(* Logix 5000 project; controller Hose_HP_Test_Rig_V1 vendor 1 type 14 code 149 rev 32.11; software revision 32.00; part 6 of 10 *)
(* tags used below, declared in another part *)
   BOTTOM_NOT_CLAMPED_STN3 : BOOL;
   FAIL_COMP_DROP_DEL : TIMER;
   FAIL_COMP_DROPPED : BOOL;
   FAIL_FLUSHED : DINT;
   FAULT_COMP_DROP_DEL : TIMER;
   FAULT_COMP_DROPPED : BOOL;
   FAULT_COMP_SENSOR : ALIAS FOR Local:2:I.Data.30;
   FAULT_FIFO_DEL : TIMER;
   FAULT_FLUSHED : DINT;
   FIFO_INDEX : DINT;
   FLUSH_BIN_DROP : TIMER;
   FLUSH_FAIL_BIN_DROP : TIMER;
   GET_FIRST_FAULTED : DINT;
   GOTO_FAIL_BIN_STN1 : DINT;
   GOTO_FAULT_BIN_STN3 : DINT;
   GOTO_FAULT_BIN_STN4 : DINT;
   ONS_100 : BOOL;
   ONS_101 : BOOL;
   ONS_102 : BOOL;
   ONS_70 : BOOL;
   ONS_76 : BOOL;
   ONS_77 : BOOL;
   ONS_78 : BOOL;
   ONS_79 : BOOL;
   ONS_80 : BOOL;
   ONS_81 : BOOL;
   ONS_82 : BOOL;
   ONS_83 : BOOL;
   ONS_84 : BOOL;
   ONS_85 : BOOL;
   ONS_86 : BOOL;
   ONS_87 : BOOL;
   ONS_88 : BOOL;
   ONS_89 : BOOL;
   ONS_90 : BOOL;
   ONS_91 : BOOL;
   ONS_92 : BOOL;
   ONS_93 : BOOL;
   ONS_95 : BOOL;
   ONS_96 : BOOL;
   ONS_97 : BOOL;
   ONS_98 : BOOL;
   ONS_99 : BOOL;
   TOP_NOT_CLAMPED_STN2 : BOOL;
   TOP_NOT_CLAMPED_STN3 : BOOL;
   TOP_NOT_CLAMPED_STN4 : BOOL;
   AUTO_TEST_ON_STN2 : BOOL;
   AUTO_TEST_ON_STN3 : BOOL;
   AUTO_TEST_ON_STN4 : BOOL;
   AUTO_TEST_SEL_STN1 : BOOL;
   AUTO_TEST_SEL_STN2 : BOOL;
   AUTO_TEST_SEL_STN3 : BOOL;
   AUTO_TEST_SEL_STN4 : BOOL;
   BOTTOM_CLAMP_2BPR_HIGH : BOOL;
   BOTTOM_CLAMP_2BPR_LOW : BOOL;
   BOTTOM_CLAMP_4BPR_HIGH : BOOL;
   BOTTOM_CLAMP_4BPR_LOW : BOOL;
   BOTTOM_CLAMP_4BPR_LOW_STN2 : BOOL;
   BOTTOM_CLAMP_PS_STN1 : ALIAS FOR Local:1:I.Data.13;
   BOTTOM_CLAMP_PS_STN2 : ALIAS FOR Local:2:I.Data.2;
   BOTTOM_CLAMP_PS_STN3 : ALIAS FOR Local:2:I.Data.7;
   BOTTOM_CLAMP_PS_STN4 : ALIAS FOR Local:2:I.Data.12;
   BOTTOM_NOT_CLAMPED_STN2 : BOOL;
   BOTTOM_NOT_CLAMPED_STN4 : BOOL;
   CHECK_TRACE_STS_STN2 : BOOL;
   CHECK_TRACE_STS_STN3 : BOOL;
   CHECK_TRACE_STS_STN4 : BOOL;
   COMP_FAULT_STN1 : BOOL;
   COMP_FAULT_STN2 : BOOL;
   COMP_FAULT_STN3 : BOOL;
   COMP_FAULT_STN4 : BOOL;
   CONS_FAIL_COUNT_STN1 : DINT;
   CONS_FAIL_COUNT_STN2 : DINT;
   CONS_FAIL_COUNT_STN3 : DINT;
   CONS_FAIL_COUNT_STN4 : DINT;
   CONS_FAIL_COUNTER_STN1 : COUNTER;
   CONS_FAIL_COUNTER_STN2 : COUNTER;
   CONS_FAIL_COUNTER_STN3 : COUNTER;
   CONS_FAIL_COUNTER_STN4 : COUNTER;
   CONS_FILL_HIGH_STN2 : BOOL;
   CONS_FILL_HIGH_STN3 : BOOL;
   CONS_FILL_HIGH_STN4 : BOOL;
   CONS_FILL_LOW_STN2 : BOOL;
   CONS_FILL_LOW_STN3 : BOOL;
   CONS_FILL_LOW_STN4 : BOOL;
   CONS_TEST_ON : BOOL;
   CONSTRICTION_CALB_SEL_STN1 : BOOL;
   CONSTRICTION_CALB_SEL_STN2 : BOOL;
   CONSTRICTION_CALB_SEL_STN3 : BOOL;
   CONSTRICTION_CALB_SEL_STN4 : BOOL;
   CONSTRICTION_NOK_STN2 : BOOL;
   CONSTRICTION_NOK_STN3 : BOOL;
   CONSTRICTION_NOK_STN4 : BOOL;
   CONSTRICTION_TEST_ON_STN1 : BOOL;
   CONSTRICTION_TEST_ON_STN2 : BOOL;
   CONSTRICTION_TEST_ON_STN3 : BOOL;
   CONSTRICTION_TEST_ON_STN4 : BOOL;
   DOOR_CLOSE_ABORT_STN2 : BOOL;
   DOOR_CLOSE_ABORT_STN3 : BOOL;
   DOOR_CLOSE_ABORT_STN4 : BOOL;
   DOOR_NOT_CLOSED_STN2 : BOOL;
   DOOR_NOT_CLOSED_STN3 : BOOL;
   DOOR_NOT_CLOSED_STN4 : BOOL;
   DOOR_NOT_OPEN_STN2 : BOOL;
   DOOR_NOT_OPEN_STN3 : BOOL;
   DOOR_NOT_OPEN_STN4 : BOOL;
   DOOR_OPEN_RS_STN1 : ALIAS FOR Local:1:I.Data.10;
   DOOR_OPEN_RS_STN2 : ALIAS FOR Local:1:I.Data.15;
   DOOR_OPEN_RS_STN3 : ALIAS FOR Local:2:I.Data.4;
   DOOR_OPEN_RS_STN4 : ALIAS FOR Local:2:I.Data.10;
   DROP_NOK_STN2 : BOOL;
   DROP_NOK_STN3 : BOOL;
   DROP_NOK_STN4 : BOOL;
   DUPLICATE_STN2 : BOOL;
   DUPLICATE_STN3 : BOOL;
   DUPLICATE_STN4 : BOOL;
   EC_STN2 : DINT;
   EC_STN3 : DINT;
   EMG_FAULTED_STN1 : BOOL;
   FAIL_ARRAY : DINT[4];
   FAIL_BIN_DOOR_PROXY : ALIAS FOR Local:2:I.Data.29;
   FAIL_COMP_SENSOR : ALIAS FOR Local:2:I.Data.25;
   FAIL_COUNT_RETEST : DINT;
   FAIL_COUNT_RETEST_STN2 : DINT;
   FAIL_COUNT_STN1 : DINT;
   FAIL_COUNT_STN2 : DINT;
   FAIL_COUNT_STN3 : DINT;
   FAIL_COUNT_STN4 : DINT;
   FAIL_COUNTER_RETEST : COUNTER;
   FAIL_COUNTER_RETEST_STN2 : COUNTER;
   FAIL_COUNTER_STN1 : COUNTER;
   FAIL_COUNTER_STN2 : COUNTER;
   FAIL_COUNTER_STN3 : COUNTER;
   FAIL_COUNTER_STN4 : COUNTER;
   FAIL_FIFO_DEL : TIMER;
   FAIL_FIFO_INDEX : DINT;
   FAIL_FIFO_STN1 : BOOL;
   FAIL_FIFO_STN2 : BOOL;
   FAIL_FIFO_STN3 : BOOL;
   FAIL_FIFO_STN4 : BOOL;
   FAIL_R1 : CONTROL;
   FAIL_RST_KS : ALIAS FOR Local:2:I.Data.14;
   FAILED_STN1 : BOOL;
   FAILED_STN2 : BOOL;
   FAILED_STN3 : BOOL;
   FAILED_STN4 : BOOL;
   FAULT_ARRAY : DINT[4];
   FAULT_COUNT_STN2 : DINT;
   FAULT_COUNT_STN3 : DINT;
   FAULT_COUNT_STN4 : DINT;
   FAULT_COUNTER_STN2 : COUNTER;
   FAULT_COUNTER_STN3 : COUNTER;
   FAULT_COUNTER_STN4 : COUNTER;
   FAULT_FIFO_STN1 : BOOL;
   FAULT_FIFO_STN2 : BOOL;
   FAULT_FIFO_STN3 : BOOL;
   FAULT_FIFO_STN4 : BOOL;
   FAULT_R1 : CONTROL;
   FAULTED_STN1 : BOOL;
   FAULTED_STN2 : BOOL;
   FAULTED_STN3 : BOOL;
   FAULTED_STN4 : BOOL;
   FILL_HIGH_STN2 : BOOL;
   FILL_HIGH_STN3 : BOOL;
   FILL_HIGH_STN4 : BOOL;
   FILL_LOW_STN2 : BOOL;
   FILL_LOW_STN3 : BOOL;
   FILL_LOW_STN4 : BOOL;
   FLT_CLR_ONS_STN2 : BOOL;
   FLT_CLR_ONS_STN3 : BOOL;
   FLT_CLR_ONS_STN4 : BOOL;
   FLT_RST_PB_STN1 : ALIAS FOR Local:1:I.Data.7;
   FLT_RST_PB_STN2 : ALIAS FOR Local:1:I.Data.8;
   FLT_RST_PB_STN3 : ALIAS FOR Local:1:I.Data.9;
   FLT_RST_PB_STN4 : ALIAS FOR Local:2:I.Data.15;
   GET_FIRST_FAILED : DINT;
   GOTO_FAIL_BIN_STN2 : DINT;
   GOTO_FAIL_BIN_STN3 : DINT;
   GOTO_FAIL_BIN_STN4 : DINT;
   GOTO_FAULT_BIN_STN2 : DINT;
   HOME_COND_NOK_STN1 : BOOL;
   HOME_COND_NOK_STN2 : BOOL;
   HOME_COND_NOK_STN3 : BOOL;
   HOME_COND_NOK_STN4 : BOOL;
   HOME_COND_OK_STN1 : BOOL;
   HOME_COND_OK_STN2 : BOOL;
   HOME_COND_OK_STN3 : BOOL;
   HOME_COND_OK_STN4 : BOOL;
   INCORRECT_STN2 : BOOL;
   INCORRECT_STN3 : BOOL;
   INCORRECT_STN4 : BOOL;
   INDV_CTEST_SEL_STN1 : BOOL;
   INDV_CTEST_SEL_STN2 : BOOL;
   INDV_CTEST_SEL_STN3 : BOOL;
   INDV_CTEST_SEL_STN4 : BOOL;
   INDV_LTEST_SEL_STN1 : BOOL;
   INDV_LTEST_SEL_STN2 : BOOL;
   INDV_LTEST_SEL_STN3 : BOOL;
   INDV_LTEST_SEL_STN4 : BOOL;
   INLET_AIR_LOW : TIMER;
   MSG_STN1 : DINT;
   MSG_STN2 : DINT;
   MSG_STN3 : DINT;
   MSG_STN4 : DINT;
   NO_COMP_FAULT_STN2 : BOOL;
   NO_COMP_FAULT_STN3 : BOOL;
   NO_COMP_FAULT_STN4 : BOOL;
   NO_SYSTEM_FAULT_STN2 : BOOL;
   NO_SYSTEM_FAULT_STN3 : BOOL;
   NO_SYSTEM_FAULT_STN4 : BOOL;
   NOT_FAILED_STN1 : BOOL;
   NOT_FAILED_STN2 : BOOL;
   NOT_FAILED_STN3 : BOOL;
   NOT_FAILED_STN4 : BOOL;
   PASS_BIN_COUNT : DINT;
   PASS_BIN_FULL : DINT;
   PASS_COUNT_STN1 : DINT;
   PASS_COUNT_STN2 : DINT;
   PASS_COUNT_STN3 : DINT;
   PASS_COUNT_STN4 : DINT;
   RETEST : BOOL;
   RST_SEQ_ON_STN1 : BOOL;
   RST_SEQ_ON_STN2 : BOOL;
   RST_SEQ_ON_STN3 : BOOL;
   RST_SEQ_ON_STN4 : BOOL;
   SCR_STS : DINT[6];
   STAB_HIGH_STN2 : BOOL;
   STAB_HIGH_STN3 : BOOL;
   STAB_HIGH_STN4 : BOOL;
   STAB_LOW_STN2 : BOOL;
   STAB_LOW_STN3 : BOOL;
   STAB_LOW_STN4 : BOOL;
   STAMP_HL : REAL;
   STAMP_LL : REAL;
   STAMP_NOT_FWD_STN2 : BOOL;
   STAMP_NOT_FWD_STN3 : BOOL;
   STAMP_NOT_FWD_STN4 : BOOL;
   STAMP_NOT_RET_STN2 : BOOL;
   STAMP_NOT_RET_STN3 : BOOL;
   STAMP_NOT_RET_STN4 : BOOL;
   STAMP_PR : REAL;
   STAMP_PR_DEL : TIMER;
   STAMP_PR_HIGH_STN2 : BOOL;
   STAMP_PR_HIGH_STN3 : BOOL;
   STAMP_PR_HIGH_STN4 : BOOL;
   STAMP_PR_LOW_STN2 : BOOL;
   STAMP_PR_LOW_STN3 : BOOL;
   STAMP_PR_LOW_STN4 : BOOL;
   STAMP_PS_STN1 : ALIAS FOR Local:1:I.Data.14;
   STAMP_PS_STN2 : ALIAS FOR Local:2:I.Data.3;
(* MainProgram, continued *)

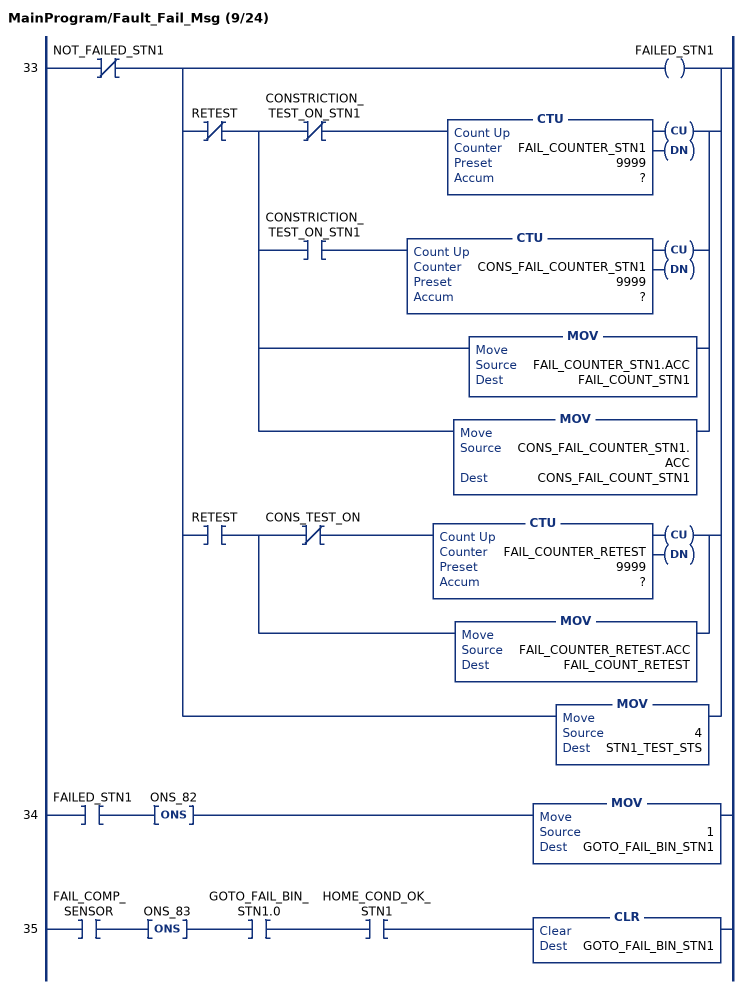
   [picture p92: MainProgram/Fault_Fail_Msg rungs 33-35]
   33: XIO(NOT_FAILED_STN1)[OTE(FAILED_STN1) ,XIO(RETEST) [XIO(CONSTRICTION_TEST_ON_STN1) CTU(FAIL_COUNTER_STN1,?,?) ,XIC(CONSTRICTION_TEST_ON_STN1) CTU(CONS_FAIL_COUNTER_STN1,?,?) ,MOV(FAIL_COUNTER_STN1.ACC,FAIL_COUNT_STN1) ,MOV(CONS_FAIL_COUNTER_STN1.ACC,CONS_FAIL_COUNT_STN1) ] ,XIC(RETEST) [XIO(CONS_TEST_ON) CTU(FAIL_COUNTER_RETEST,?,?) ,MOV(FAIL_COUNTER_RETEST.ACC,FAIL_COUNT_RETEST) ] ,MOV(4,STN1_TEST_STS) ];
   34: XIC(FAILED_STN1)ONS(ONS_82)MOV(1,GOTO_FAIL_BIN_STN1);
   35: XIC(FAIL_COMP_SENSOR)ONS(ONS_83)XIC(GOTO_FAIL_BIN_STN1.0)XIC(HOME_COND_OK_STN1)CLR(GOTO_FAIL_BIN_STN1);
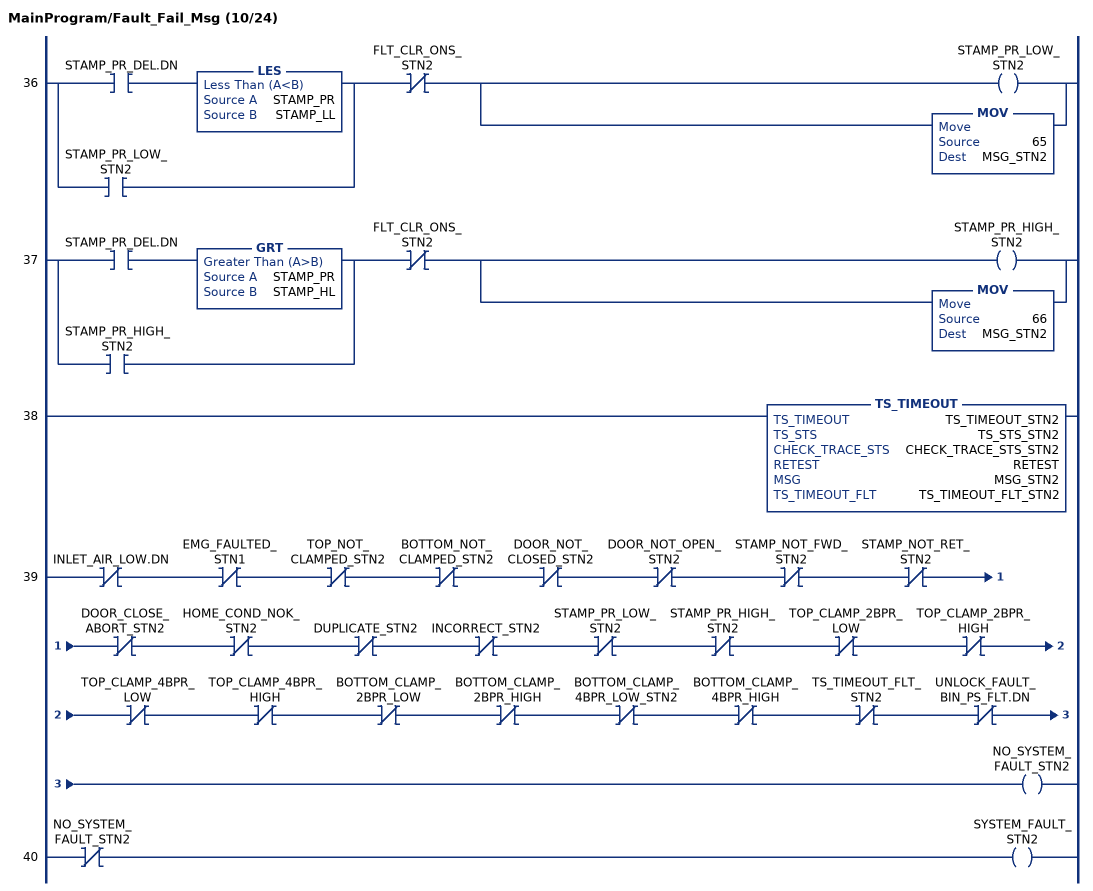
   36: [XIC(STAMP_PR_DEL.DN) LES(STAMP_PR,STAMP_LL) ,XIC(STAMP_PR_LOW_STN2) ]XIO(FLT_CLR_ONS_STN2)[OTE(STAMP_PR_LOW_STN2) ,MOV(65,MSG_STN2) ];
   37: [XIC(STAMP_PR_DEL.DN) GRT(STAMP_PR,STAMP_HL) ,XIC(STAMP_PR_HIGH_STN2) ]XIO(FLT_CLR_ONS_STN2)[OTE(STAMP_PR_HIGH_STN2) ,MOV(66,MSG_STN2) ];
   38: TS_TIMEOUT(TS_TIMEOUT_STN2,TS_STS_STN2,CHECK_TRACE_STS_STN2,RETEST,MSG_STN2,TS_TIMEOUT_FLT_STN2);
   39: XIO(INLET_AIR_LOW.DN)XIO(EMG_FAULTED_STN1)XIO(TOP_NOT_CLAMPED_STN2)XIO(BOTTOM_NOT_CLAMPED_STN2)XIO(DOOR_NOT_CLOSED_STN2)XIO(DOOR_NOT_OPEN_STN2)XIO(STAMP_NOT_FWD_STN2)XIO(STAMP_NOT_RET_STN2)XIO(DOOR_CLOSE_ABORT_STN2)XIO(HOME_COND_NOK_STN2)XIO(DUPLICATE_STN2)XIO(INCORRECT_STN2)XIO(STAMP_PR_LOW_STN2)XIO(STAMP_PR_HIGH_STN2)XIO(TOP_CLAMP_2BPR_LOW)XIO(TOP_CLAMP_2BPR_HIGH)XIO(TOP_CLAMP_4BPR_LOW)XIO(TOP_CLAMP_4BPR_HIGH)XIO(BOTTOM_CLAMP_2BPR_LOW)XIO(BOTTOM_CLAMP_2BPR_HIGH)XIO(BOTTOM_CLAMP_4BPR_LOW_STN2)XIO(BOTTOM_CLAMP_4BPR_HIGH)XIO(TS_TIMEOUT_FLT_STN2)XIO(UNLOCK_FAULT_BIN_PS_FLT.DN)OTE(NO_SYSTEM_FAULT_STN2);
   40: XIO(NO_SYSTEM_FAULT_STN2)OTE(SYSTEM_FAULT_STN2);
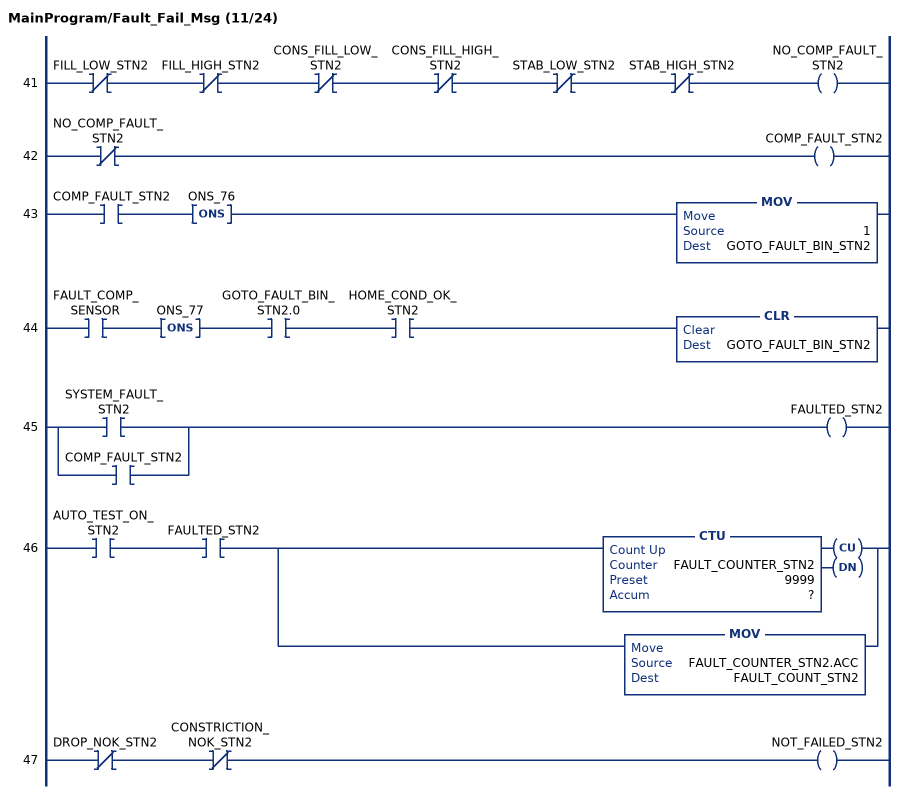
   41: XIO(FILL_LOW_STN2)XIO(FILL_HIGH_STN2)XIO(CONS_FILL_LOW_STN2)XIO(CONS_FILL_HIGH_STN2)XIO(STAB_LOW_STN2)XIO(STAB_HIGH_STN2)OTE(NO_COMP_FAULT_STN2);
   42: XIO(NO_COMP_FAULT_STN2)OTE(COMP_FAULT_STN2);
   43: XIC(COMP_FAULT_STN2)ONS(ONS_76)MOV(1,GOTO_FAULT_BIN_STN2);
   44: XIC(FAULT_COMP_SENSOR)ONS(ONS_77)XIC(GOTO_FAULT_BIN_STN2.0)XIC(HOME_COND_OK_STN2)CLR(GOTO_FAULT_BIN_STN2);
   45: [XIC(SYSTEM_FAULT_STN2) ,XIC(COMP_FAULT_STN2) ]OTE(FAULTED_STN2);
   46: XIC(AUTO_TEST_ON_STN2)XIC(FAULTED_STN2)[CTU(FAULT_COUNTER_STN2,?,?) ,MOV(FAULT_COUNTER_STN2.ACC,FAULT_COUNT_STN2) ];
   47: XIO(DROP_NOK_STN2)XIO(CONSTRICTION_NOK_STN2)OTE(NOT_FAILED_STN2);
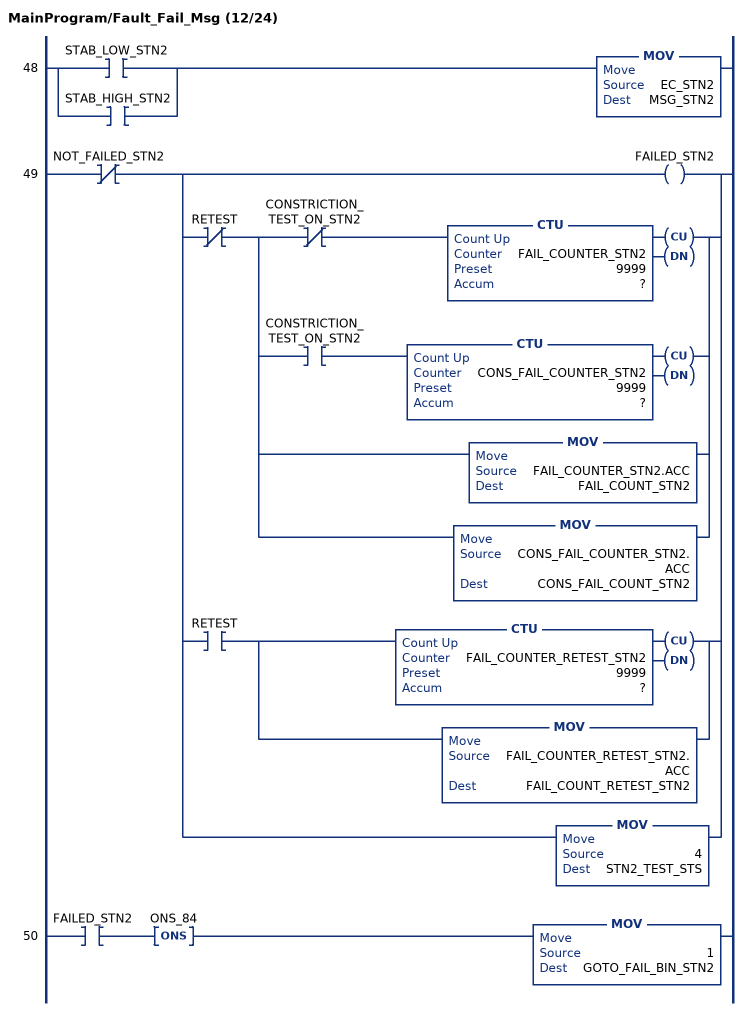
   48: [XIC(STAB_LOW_STN2) ,XIC(STAB_HIGH_STN2) ]MOV(EC_STN2,MSG_STN2);
   49: XIO(NOT_FAILED_STN2)[OTE(FAILED_STN2) ,XIO(RETEST) [[XIO(CONSTRICTION_TEST_ON_STN2) CTU(FAIL_COUNTER_STN2,?,?) ,XIC(CONSTRICTION_TEST_ON_STN2) CTU(CONS_FAIL_COUNTER_STN2,?,?) ] ,MOV(FAIL_COUNTER_STN2.ACC,FAIL_COUNT_STN2) ,MOV(CONS_FAIL_COUNTER_STN2.ACC,CONS_FAIL_COUNT_STN2) ] ,XIC(RETEST) [CTU(FAIL_COUNTER_RETEST_STN2,?,?) ,MOV(FAIL_COUNTER_RETEST_STN2.ACC,FAIL_COUNT_RETEST_STN2) ] ,MOV(4,STN2_TEST_STS) ];
   50: XIC(FAILED_STN2)ONS(ONS_84)MOV(1,GOTO_FAIL_BIN_STN2);
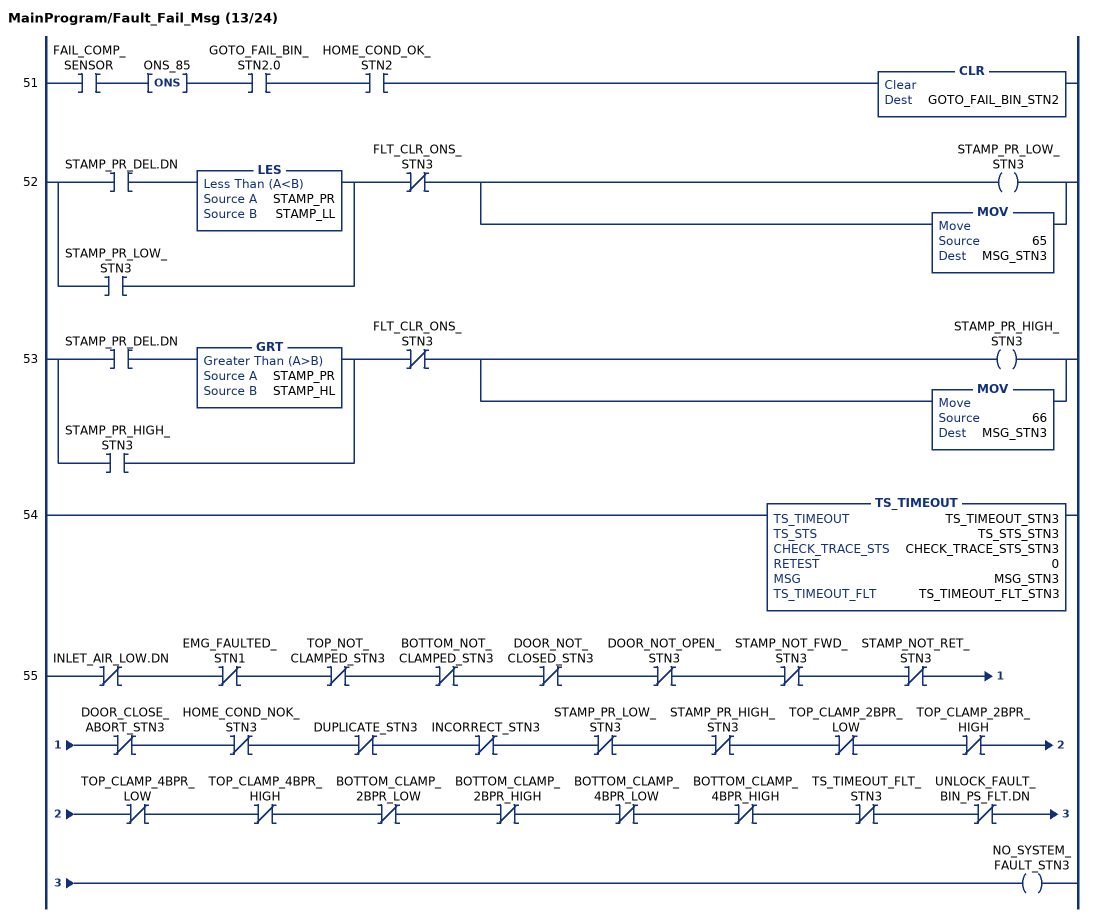
   51: XIC(FAIL_COMP_SENSOR)ONS(ONS_85)XIC(GOTO_FAIL_BIN_STN2.0)XIC(HOME_COND_OK_STN2)CLR(GOTO_FAIL_BIN_STN2);
   52: [XIC(STAMP_PR_DEL.DN) LES(STAMP_PR,STAMP_LL) ,XIC(STAMP_PR_LOW_STN3) ]XIO(FLT_CLR_ONS_STN3)[OTE(STAMP_PR_LOW_STN3) ,MOV(65,MSG_STN3) ];
   53: [XIC(STAMP_PR_DEL.DN) GRT(STAMP_PR,STAMP_HL) ,XIC(STAMP_PR_HIGH_STN3) ]XIO(FLT_CLR_ONS_STN3)[OTE(STAMP_PR_HIGH_STN3) ,MOV(66,MSG_STN3) ];
   54: TS_TIMEOUT(TS_TIMEOUT_STN3,TS_STS_STN3,CHECK_TRACE_STS_STN3,0,MSG_STN3,TS_TIMEOUT_FLT_STN3);
   55: XIO(INLET_AIR_LOW.DN)XIO(EMG_FAULTED_STN1)XIO(TOP_NOT_CLAMPED_STN3)XIO(BOTTOM_NOT_CLAMPED_STN3)XIO(DOOR_NOT_CLOSED_STN3)XIO(DOOR_NOT_OPEN_STN3)XIO(STAMP_NOT_FWD_STN3)XIO(STAMP_NOT_RET_STN3)XIO(DOOR_CLOSE_ABORT_STN3)XIO(HOME_COND_NOK_STN3)XIO(DUPLICATE_STN3)XIO(INCORRECT_STN3)XIO(STAMP_PR_LOW_STN3)XIO(STAMP_PR_HIGH_STN3)XIO(TOP_CLAMP_2BPR_LOW)XIO(TOP_CLAMP_2BPR_HIGH)XIO(TOP_CLAMP_4BPR_LOW)XIO(TOP_CLAMP_4BPR_HIGH)XIO(BOTTOM_CLAMP_2BPR_LOW)XIO(BOTTOM_CLAMP_2BPR_HIGH)XIO(BOTTOM_CLAMP_4BPR_LOW)XIO(BOTTOM_CLAMP_4BPR_HIGH)XIO(TS_TIMEOUT_FLT_STN3)XIO(UNLOCK_FAULT_BIN_PS_FLT.DN)OTE(NO_SYSTEM_FAULT_STN3);
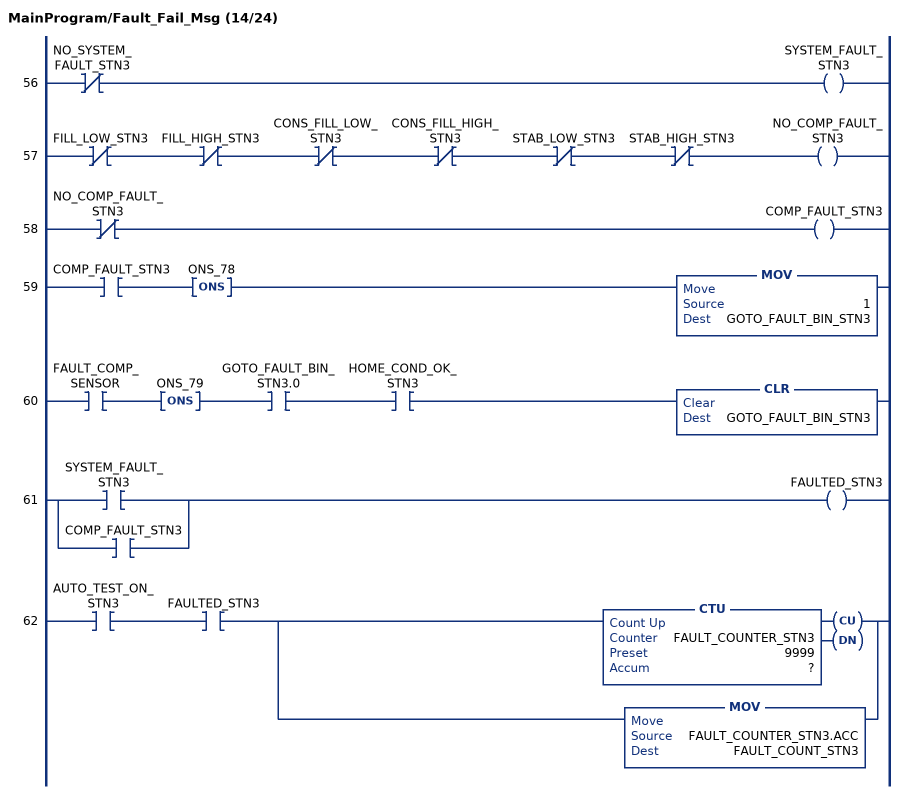
   56: XIO(NO_SYSTEM_FAULT_STN3)OTE(SYSTEM_FAULT_STN3);
   57: XIO(FILL_LOW_STN3)XIO(FILL_HIGH_STN3)XIO(CONS_FILL_LOW_STN3)XIO(CONS_FILL_HIGH_STN3)XIO(STAB_LOW_STN3)XIO(STAB_HIGH_STN3)OTE(NO_COMP_FAULT_STN3);
   58: XIO(NO_COMP_FAULT_STN3)OTE(COMP_FAULT_STN3);
   59: XIC(COMP_FAULT_STN3)ONS(ONS_78)MOV(1,GOTO_FAULT_BIN_STN3);
   60: XIC(FAULT_COMP_SENSOR)ONS(ONS_79)XIC(GOTO_FAULT_BIN_STN3.0)XIC(HOME_COND_OK_STN3)CLR(GOTO_FAULT_BIN_STN3);
   61: [XIC(SYSTEM_FAULT_STN3) ,XIC(COMP_FAULT_STN3) ]OTE(FAULTED_STN3);
   62: XIC(AUTO_TEST_ON_STN3)XIC(FAULTED_STN3)[CTU(FAULT_COUNTER_STN3,?,?) ,MOV(FAULT_COUNTER_STN3.ACC,FAULT_COUNT_STN3) ];
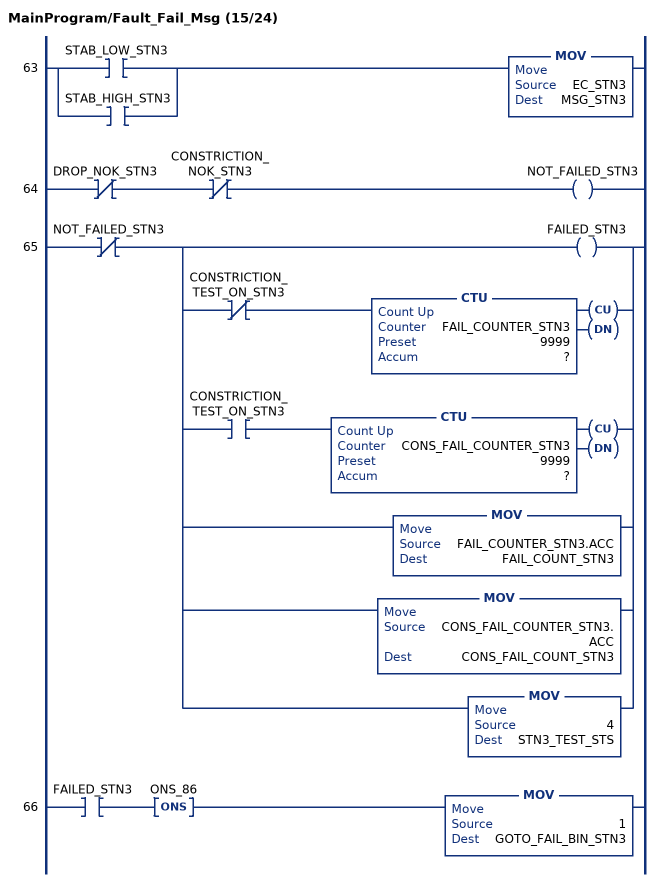
   63: [XIC(STAB_LOW_STN3) ,XIC(STAB_HIGH_STN3) ]MOV(EC_STN3,MSG_STN3);
   64: XIO(DROP_NOK_STN3)XIO(CONSTRICTION_NOK_STN3)OTE(NOT_FAILED_STN3);
   65: XIO(NOT_FAILED_STN3)[OTE(FAILED_STN3) ,XIO(CONSTRICTION_TEST_ON_STN3) CTU(FAIL_COUNTER_STN3,?,?) ,XIC(CONSTRICTION_TEST_ON_STN3) CTU(CONS_FAIL_COUNTER_STN3,?,?) ,MOV(FAIL_COUNTER_STN3.ACC,FAIL_COUNT_STN3) ,MOV(CONS_FAIL_COUNTER_STN3.ACC,CONS_FAIL_COUNT_STN3) ,MOV(4,STN3_TEST_STS) ];
   66: XIC(FAILED_STN3)ONS(ONS_86)MOV(1,GOTO_FAIL_BIN_STN3);
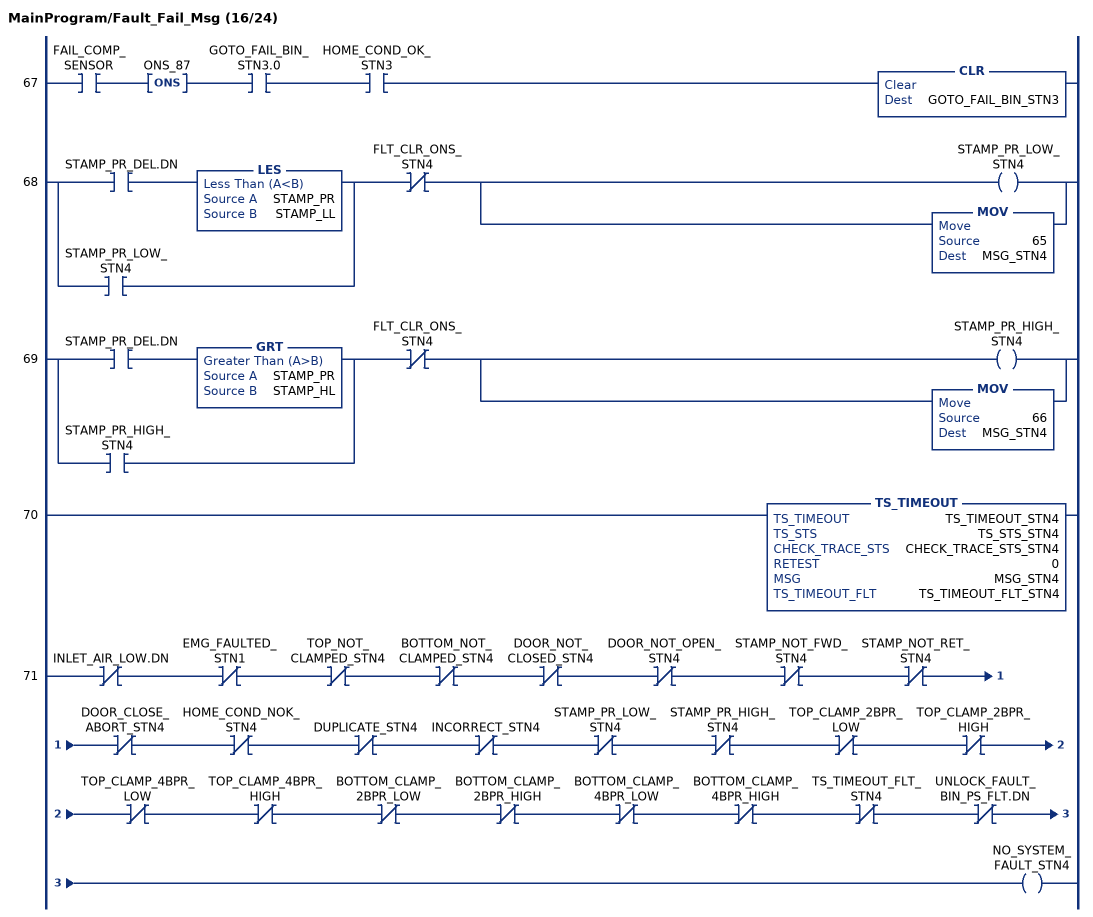
   67: XIC(FAIL_COMP_SENSOR)ONS(ONS_87)XIC(GOTO_FAIL_BIN_STN3.0)XIC(HOME_COND_OK_STN3)CLR(GOTO_FAIL_BIN_STN3);
   68: [XIC(STAMP_PR_DEL.DN) LES(STAMP_PR,STAMP_LL) ,XIC(STAMP_PR_LOW_STN4) ]XIO(FLT_CLR_ONS_STN4)[OTE(STAMP_PR_LOW_STN4) ,MOV(65,MSG_STN4) ];
   69: [XIC(STAMP_PR_DEL.DN) GRT(STAMP_PR,STAMP_HL) ,XIC(STAMP_PR_HIGH_STN4) ]XIO(FLT_CLR_ONS_STN4)[OTE(STAMP_PR_HIGH_STN4) ,MOV(66,MSG_STN4) ];
   70: TS_TIMEOUT(TS_TIMEOUT_STN4,TS_STS_STN4,CHECK_TRACE_STS_STN4,0,MSG_STN4,TS_TIMEOUT_FLT_STN4);
   71: XIO(INLET_AIR_LOW.DN)XIO(EMG_FAULTED_STN1)XIO(TOP_NOT_CLAMPED_STN4)XIO(BOTTOM_NOT_CLAMPED_STN4)XIO(DOOR_NOT_CLOSED_STN4)XIO(DOOR_NOT_OPEN_STN4)XIO(STAMP_NOT_FWD_STN4)XIO(STAMP_NOT_RET_STN4)XIO(DOOR_CLOSE_ABORT_STN4)XIO(HOME_COND_NOK_STN4)XIO(DUPLICATE_STN4)XIO(INCORRECT_STN4)XIO(STAMP_PR_LOW_STN4)XIO(STAMP_PR_HIGH_STN4)XIO(TOP_CLAMP_2BPR_LOW)XIO(TOP_CLAMP_2BPR_HIGH)XIO(TOP_CLAMP_4BPR_LOW)XIO(TOP_CLAMP_4BPR_HIGH)XIO(BOTTOM_CLAMP_2BPR_LOW)XIO(BOTTOM_CLAMP_2BPR_HIGH)XIO(BOTTOM_CLAMP_4BPR_LOW)XIO(BOTTOM_CLAMP_4BPR_HIGH)XIO(TS_TIMEOUT_FLT_STN4)XIO(UNLOCK_FAULT_BIN_PS_FLT.DN)OTE(NO_SYSTEM_FAULT_STN4);
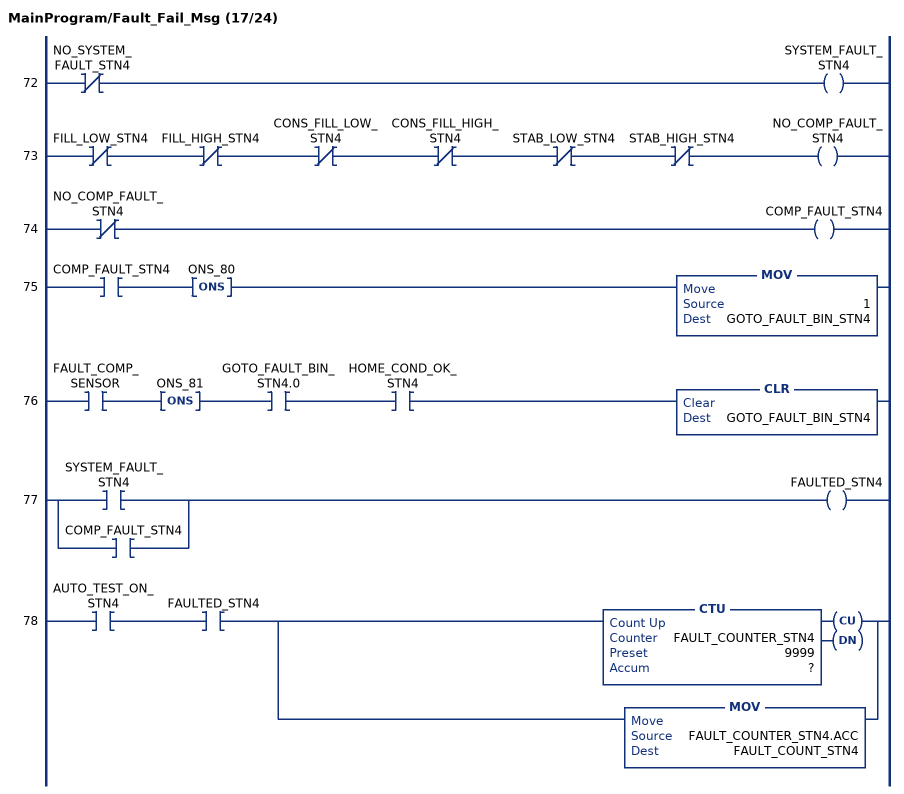
   72: XIO(NO_SYSTEM_FAULT_STN4)OTE(SYSTEM_FAULT_STN4);
   73: XIO(FILL_LOW_STN4)XIO(FILL_HIGH_STN4)XIO(CONS_FILL_LOW_STN4)XIO(CONS_FILL_HIGH_STN4)XIO(STAB_LOW_STN4)XIO(STAB_HIGH_STN4)OTE(NO_COMP_FAULT_STN4);
   74: XIO(NO_COMP_FAULT_STN4)OTE(COMP_FAULT_STN4);
   75: XIC(COMP_FAULT_STN4)ONS(ONS_80)MOV(1,GOTO_FAULT_BIN_STN4);
   76: XIC(FAULT_COMP_SENSOR)ONS(ONS_81)XIC(GOTO_FAULT_BIN_STN4.0)XIC(HOME_COND_OK_STN4)CLR(GOTO_FAULT_BIN_STN4);
   77: [XIC(SYSTEM_FAULT_STN4) ,XIC(COMP_FAULT_STN4) ]OTE(FAULTED_STN4);
   78: XIC(AUTO_TEST_ON_STN4)XIC(FAULTED_STN4)[CTU(FAULT_COUNTER_STN4,?,?) ,MOV(FAULT_COUNTER_STN4.ACC,FAULT_COUNT_STN4) ];
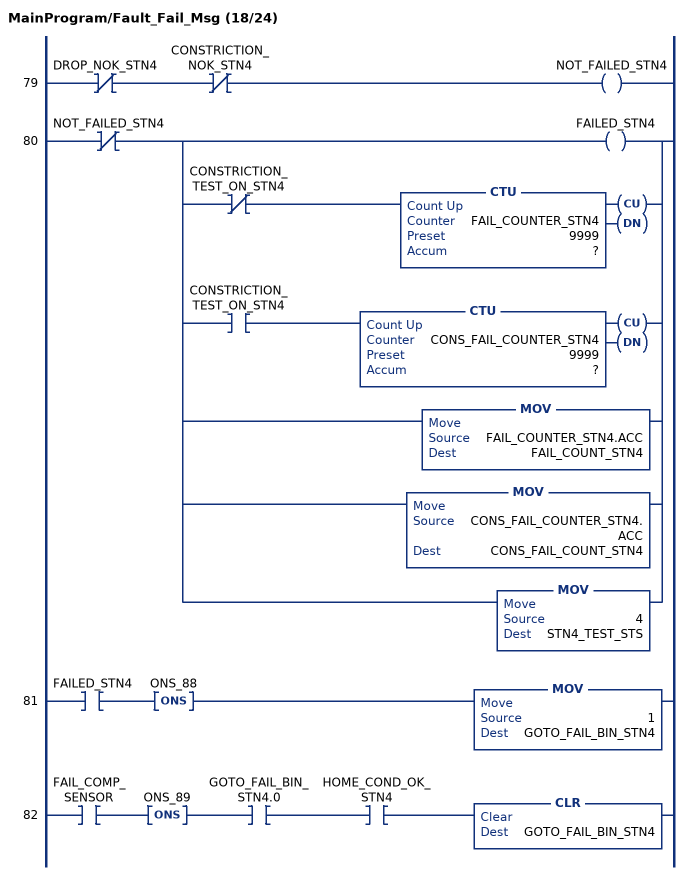
   79: XIO(DROP_NOK_STN4)XIO(CONSTRICTION_NOK_STN4)OTE(NOT_FAILED_STN4);
   80: XIO(NOT_FAILED_STN4)[OTE(FAILED_STN4) ,XIO(CONSTRICTION_TEST_ON_STN4) CTU(FAIL_COUNTER_STN4,?,?) ,XIC(CONSTRICTION_TEST_ON_STN4) CTU(CONS_FAIL_COUNTER_STN4,?,?) ,MOV(FAIL_COUNTER_STN4.ACC,FAIL_COUNT_STN4) ,MOV(CONS_FAIL_COUNTER_STN4.ACC,CONS_FAIL_COUNT_STN4) ,MOV(4,STN4_TEST_STS) ];
   81: XIC(FAILED_STN4)ONS(ONS_88)MOV(1,GOTO_FAIL_BIN_STN4);
   82: XIC(FAIL_COMP_SENSOR)ONS(ONS_89)XIC(GOTO_FAIL_BIN_STN4.0)XIC(HOME_COND_OK_STN4)CLR(GOTO_FAIL_BIN_STN4);
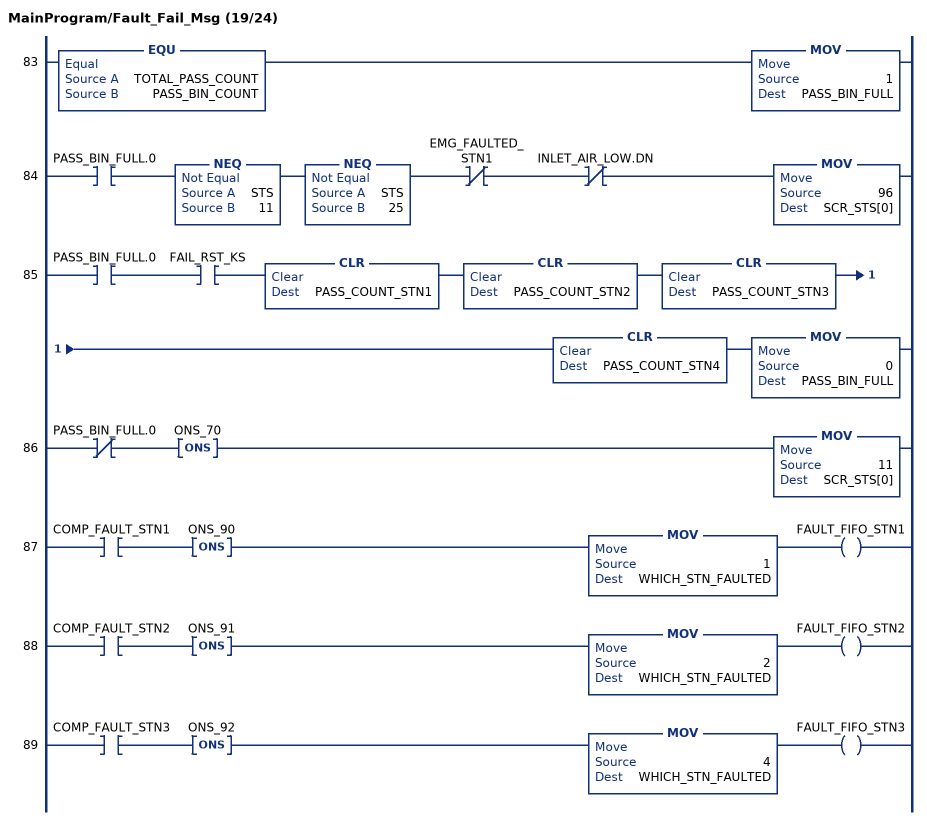
   83: EQU(TOTAL_PASS_COUNT,PASS_BIN_COUNT)MOV(1,PASS_BIN_FULL);
   84: XIC(PASS_BIN_FULL.0)NEQ(STS,11)NEQ(STS,25)XIO(EMG_FAULTED_STN1)XIO(INLET_AIR_LOW.DN)MOV(96,SCR_STS[0]);
   85: XIC(PASS_BIN_FULL.0)XIC(FAIL_RST_KS)CLR(PASS_COUNT_STN1)CLR(PASS_COUNT_STN2)CLR(PASS_COUNT_STN3)CLR(PASS_COUNT_STN4)MOV(0,PASS_BIN_FULL);
   86: XIO(PASS_BIN_FULL.0)ONS(ONS_70)MOV(11,SCR_STS[0]);
   87: XIC(COMP_FAULT_STN1)ONS(ONS_90)MOV(1,WHICH_STN_FAULTED)OTE(FAULT_FIFO_STN1);
   88: XIC(COMP_FAULT_STN2)ONS(ONS_91)MOV(2,WHICH_STN_FAULTED)OTE(FAULT_FIFO_STN2);
   89: XIC(COMP_FAULT_STN3)ONS(ONS_92)MOV(4,WHICH_STN_FAULTED)OTE(FAULT_FIFO_STN3);
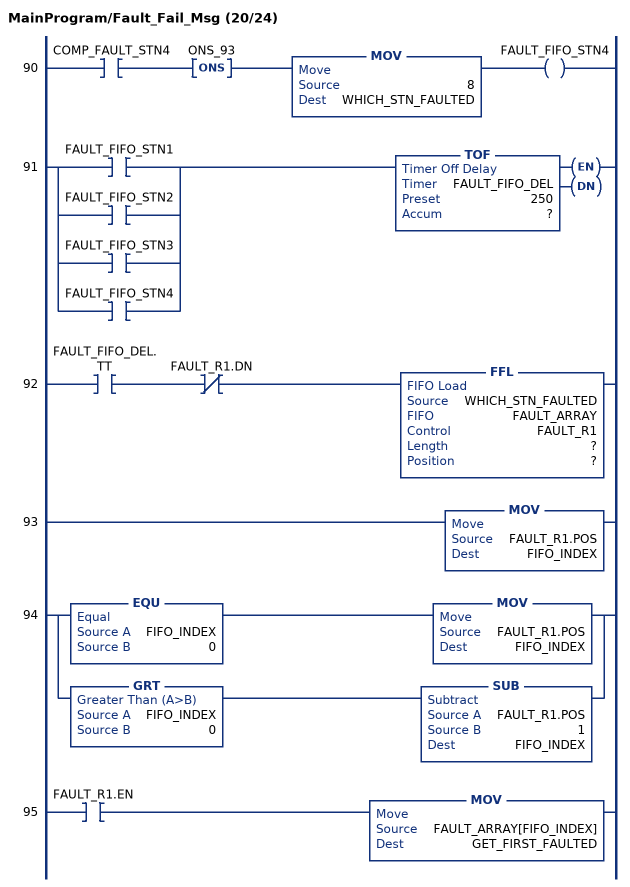
   90: XIC(COMP_FAULT_STN4)ONS(ONS_93)MOV(8,WHICH_STN_FAULTED)OTE(FAULT_FIFO_STN4);
   91: [XIC(FAULT_FIFO_STN1) ,XIC(FAULT_FIFO_STN2) ,XIC(FAULT_FIFO_STN3) ,XIC(FAULT_FIFO_STN4) ]TOF(FAULT_FIFO_DEL,?,?);
   92: XIC(FAULT_FIFO_DEL.TT)XIO(FAULT_R1.DN)FFL(WHICH_STN_FAULTED,FAULT_ARRAY,FAULT_R1,?,?);
   93: MOV(FAULT_R1.POS,FIFO_INDEX);
   94: [EQU(FIFO_INDEX,0) MOV(FAULT_R1.POS,FIFO_INDEX) ,GRT(FIFO_INDEX,0) SUB(FAULT_R1.POS,1,FIFO_INDEX) ];
   95: XIC(FAULT_R1.EN)MOV(FAULT_ARRAY[FIFO_INDEX],GET_FIRST_FAULTED);
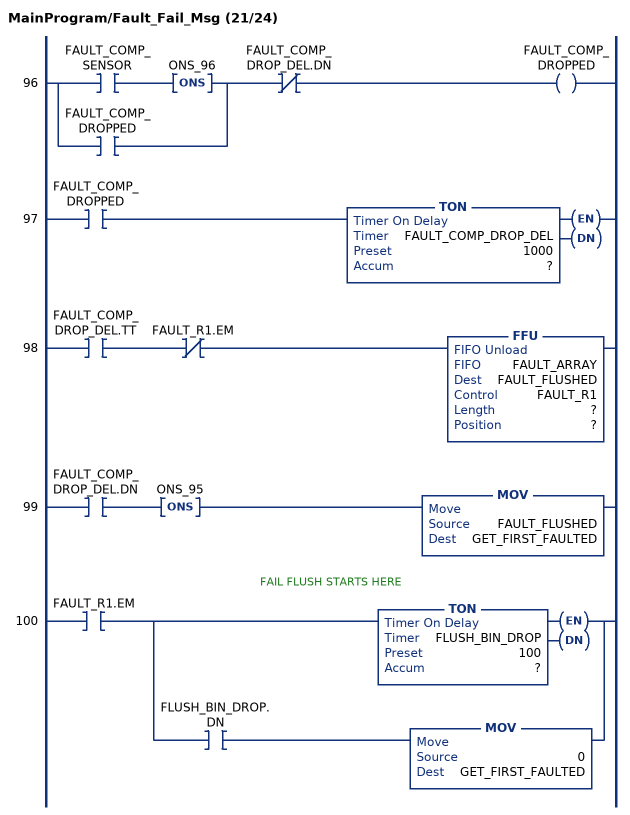
   96: [XIC(FAULT_COMP_SENSOR) ONS(ONS_96) ,XIC(FAULT_COMP_DROPPED) ]XIO(FAULT_COMP_DROP_DEL.DN)OTE(FAULT_COMP_DROPPED);
   97: XIC(FAULT_COMP_DROPPED)TON(FAULT_COMP_DROP_DEL,?,?);
   98: XIC(FAULT_COMP_DROP_DEL.TT)XIO(FAULT_R1.EM)FFU(FAULT_ARRAY,FAULT_FLUSHED,FAULT_R1,?,?);
   99: XIC(FAULT_COMP_DROP_DEL.DN)ONS(ONS_95)MOV(FAULT_FLUSHED,GET_FIRST_FAULTED);
   // FAIL FLUSH STARTS HERE
   100: XIC(FAULT_R1.EM)[TON(FLUSH_BIN_DROP,?,?) ,XIC(FLUSH_BIN_DROP.DN) MOV(0,GET_FIRST_FAULTED) ];
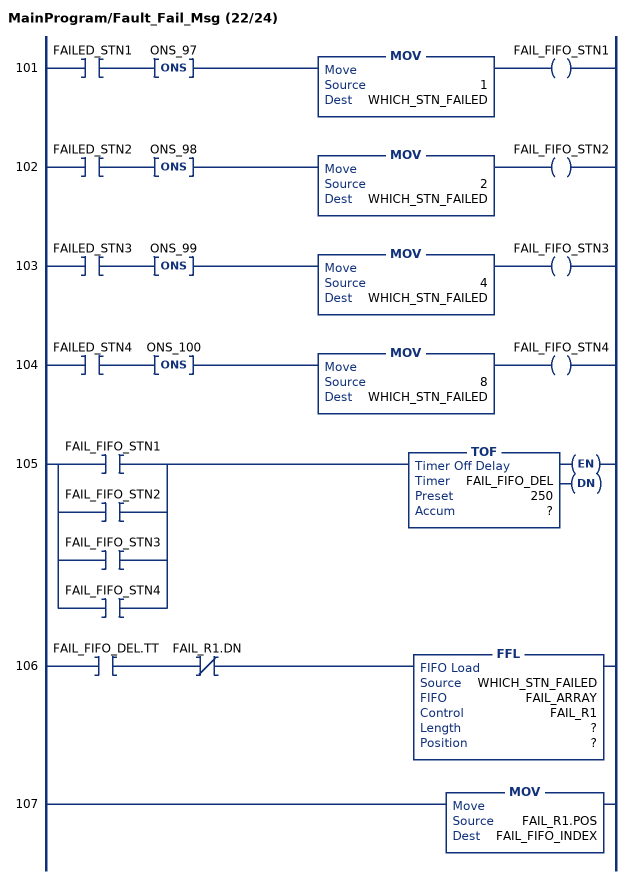
   101: XIC(FAILED_STN1)ONS(ONS_97)MOV(1,WHICH_STN_FAILED)OTE(FAIL_FIFO_STN1);
   102: XIC(FAILED_STN2)ONS(ONS_98)MOV(2,WHICH_STN_FAILED)OTE(FAIL_FIFO_STN2);
   103: XIC(FAILED_STN3)ONS(ONS_99)MOV(4,WHICH_STN_FAILED)OTE(FAIL_FIFO_STN3);
   104: XIC(FAILED_STN4)ONS(ONS_100)MOV(8,WHICH_STN_FAILED)OTE(FAIL_FIFO_STN4);
   105: [XIC(FAIL_FIFO_STN1) ,XIC(FAIL_FIFO_STN2) ,XIC(FAIL_FIFO_STN3) ,XIC(FAIL_FIFO_STN4) ]TOF(FAIL_FIFO_DEL,?,?);
   106: XIC(FAIL_FIFO_DEL.TT)XIO(FAIL_R1.DN)FFL(WHICH_STN_FAILED,FAIL_ARRAY,FAIL_R1,?,?);
   107: MOV(FAIL_R1.POS,FAIL_FIFO_INDEX);
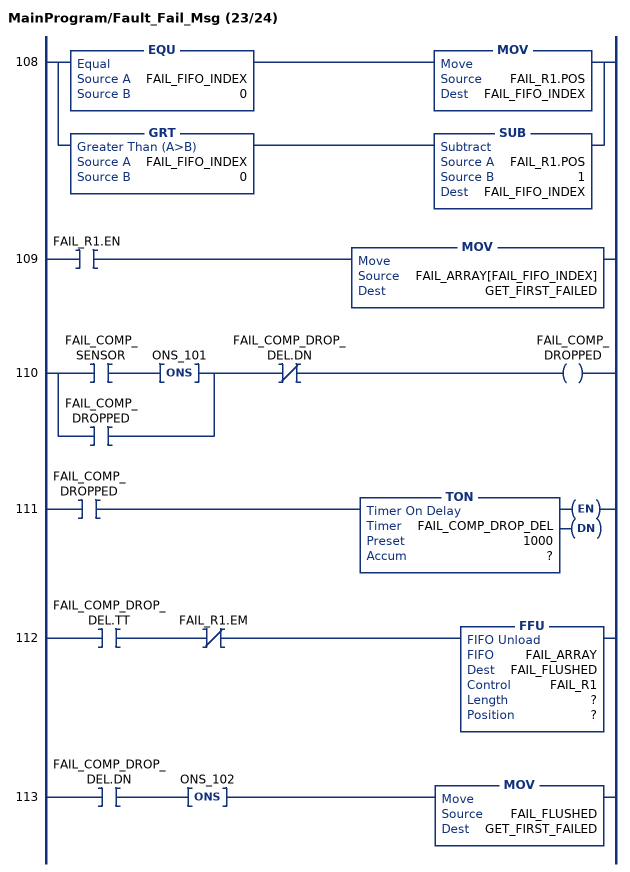
   108: [EQU(FAIL_FIFO_INDEX,0) MOV(FAIL_R1.POS,FAIL_FIFO_INDEX) ,GRT(FAIL_FIFO_INDEX,0) SUB(FAIL_R1.POS,1,FAIL_FIFO_INDEX) ];
   109: XIC(FAIL_R1.EN)MOV(FAIL_ARRAY[FAIL_FIFO_INDEX],GET_FIRST_FAILED);
   110: [XIC(FAIL_COMP_SENSOR) ONS(ONS_101) ,XIC(FAIL_COMP_DROPPED) ]XIO(FAIL_COMP_DROP_DEL.DN)OTE(FAIL_COMP_DROPPED);
   111: XIC(FAIL_COMP_DROPPED)TON(FAIL_COMP_DROP_DEL,?,?);
   112: XIC(FAIL_COMP_DROP_DEL.TT)XIO(FAIL_R1.EM)FFU(FAIL_ARRAY,FAIL_FLUSHED,FAIL_R1,?,?);
   113: XIC(FAIL_COMP_DROP_DEL.DN)ONS(ONS_102)MOV(FAIL_FLUSHED,GET_FIRST_FAILED);
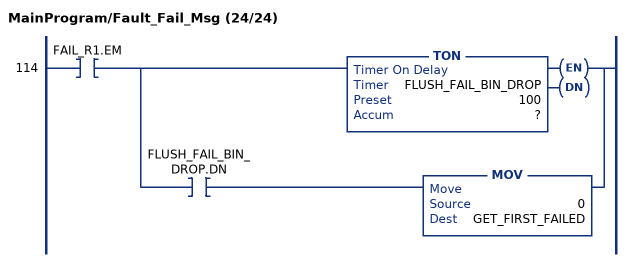
   114: XIC(FAIL_R1.EM)[TON(FLUSH_FAIL_BIN_DROP,?,?) ,XIC(FLUSH_FAIL_BIN_DROP.DN) MOV(0,GET_FIRST_FAILED) ];
END_ROUTINE

ROUTINE Home_Cond_Check   (* ladder *)
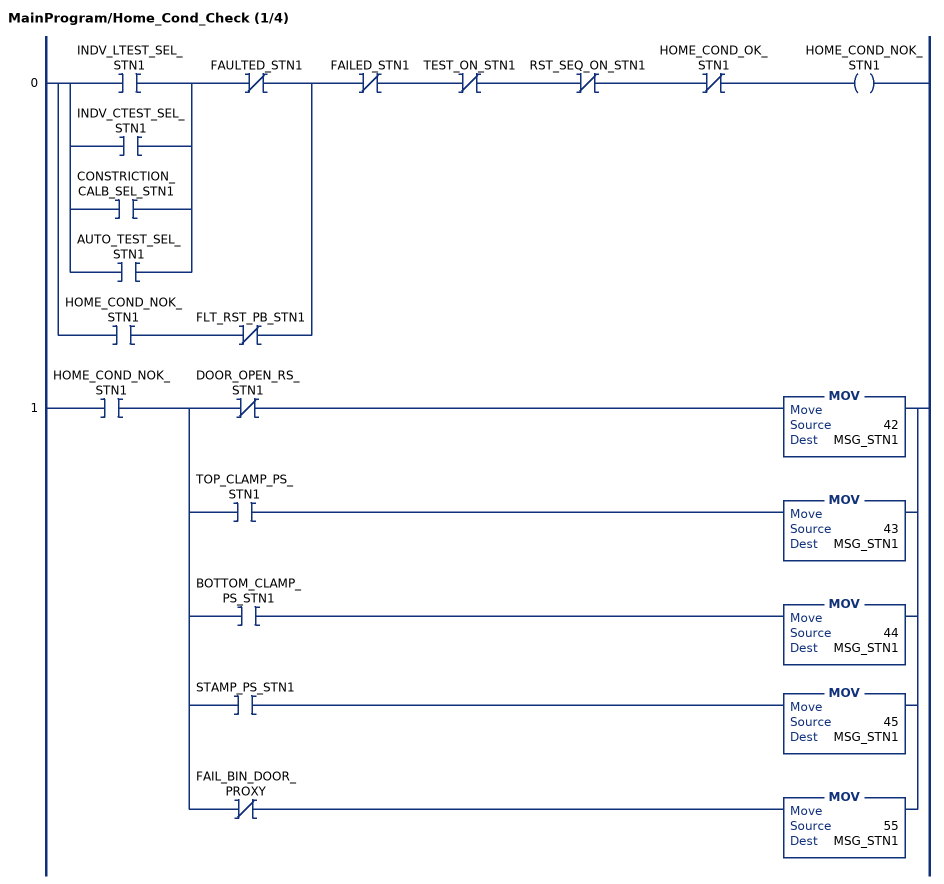
   0: [[XIC(INDV_LTEST_SEL_STN1) ,XIC(INDV_CTEST_SEL_STN1) ,XIC(CONSTRICTION_CALB_SEL_STN1) ,XIC(AUTO_TEST_SEL_STN1) ] XIO(FAULTED_STN1) ,XIC(HOME_COND_NOK_STN1) XIO(FLT_RST_PB_STN1) ]XIO(FAILED_STN1)XIO(TEST_ON_STN1)XIO(RST_SEQ_ON_STN1)XIO(HOME_COND_OK_STN1)OTE(HOME_COND_NOK_STN1);
   1: XIC(HOME_COND_NOK_STN1)[XIO(DOOR_OPEN_RS_STN1) MOV(42,MSG_STN1) ,XIC(TOP_CLAMP_PS_STN1) MOV(43,MSG_STN1) ,XIC(BOTTOM_CLAMP_PS_STN1) MOV(44,MSG_STN1) ,XIC(STAMP_PS_STN1) MOV(45,MSG_STN1) ,XIO(FAIL_BIN_DOOR_PROXY) MOV(55,MSG_STN1) ];
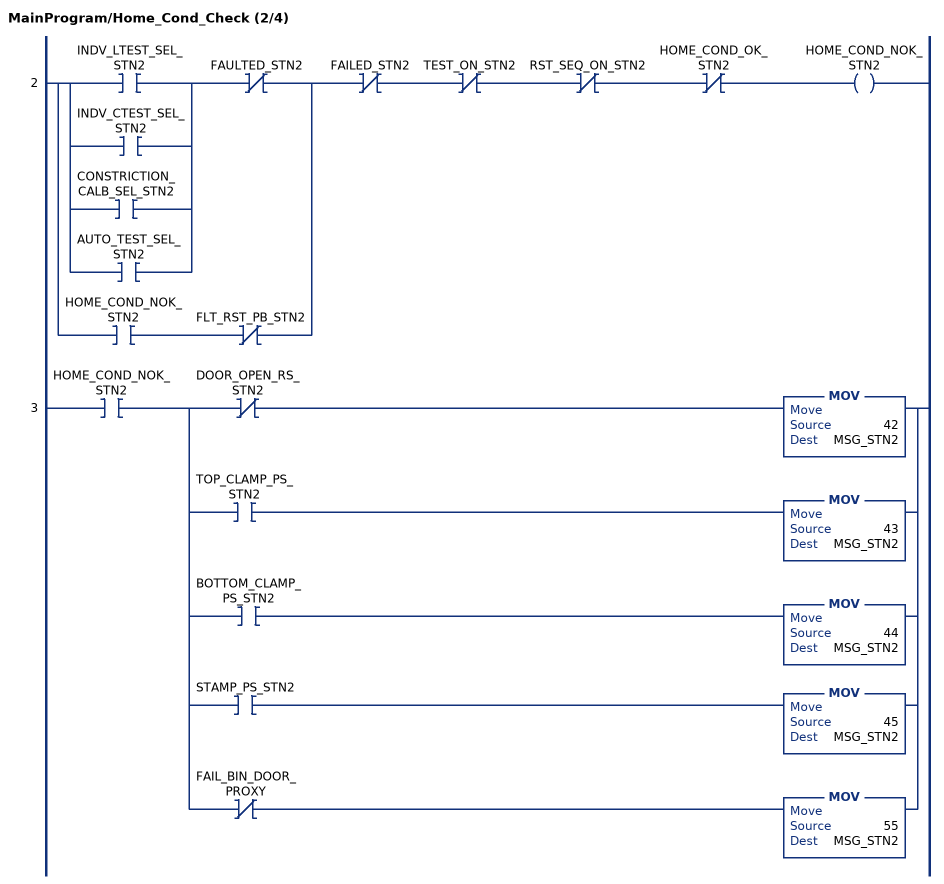
   2: [[XIC(INDV_LTEST_SEL_STN2) ,XIC(INDV_CTEST_SEL_STN2) ,XIC(CONSTRICTION_CALB_SEL_STN2) ,XIC(AUTO_TEST_SEL_STN2) ] XIO(FAULTED_STN2) ,XIC(HOME_COND_NOK_STN2) XIO(FLT_RST_PB_STN2) ]XIO(FAILED_STN2)XIO(TEST_ON_STN2)XIO(RST_SEQ_ON_STN2)XIO(HOME_COND_OK_STN2)OTE(HOME_COND_NOK_STN2);
   3: XIC(HOME_COND_NOK_STN2)[XIO(DOOR_OPEN_RS_STN2) MOV(42,MSG_STN2) ,XIC(TOP_CLAMP_PS_STN2) MOV(43,MSG_STN2) ,XIC(BOTTOM_CLAMP_PS_STN2) MOV(44,MSG_STN2) ,XIC(STAMP_PS_STN2) MOV(45,MSG_STN2) ,XIO(FAIL_BIN_DOOR_PROXY) MOV(55,MSG_STN2) ];
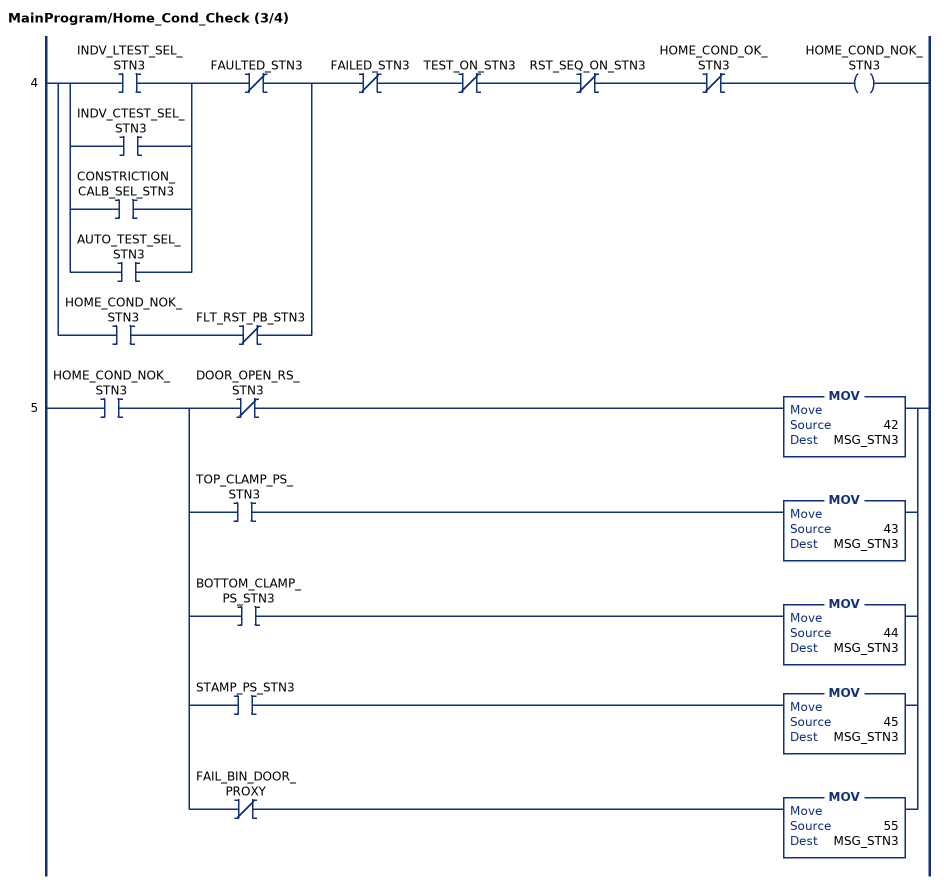
   4: [[XIC(INDV_LTEST_SEL_STN3) ,XIC(INDV_CTEST_SEL_STN3) ,XIC(CONSTRICTION_CALB_SEL_STN3) ,XIC(AUTO_TEST_SEL_STN3) ] XIO(FAULTED_STN3) ,XIC(HOME_COND_NOK_STN3) XIO(FLT_RST_PB_STN3) ]XIO(FAILED_STN3)XIO(TEST_ON_STN3)XIO(RST_SEQ_ON_STN3)XIO(HOME_COND_OK_STN3)OTE(HOME_COND_NOK_STN3);
   5: XIC(HOME_COND_NOK_STN3)[XIO(DOOR_OPEN_RS_STN3) MOV(42,MSG_STN3) ,XIC(TOP_CLAMP_PS_STN3) MOV(43,MSG_STN3) ,XIC(BOTTOM_CLAMP_PS_STN3) MOV(44,MSG_STN3) ,XIC(STAMP_PS_STN3) MOV(45,MSG_STN3) ,XIO(FAIL_BIN_DOOR_PROXY) MOV(55,MSG_STN3) ];
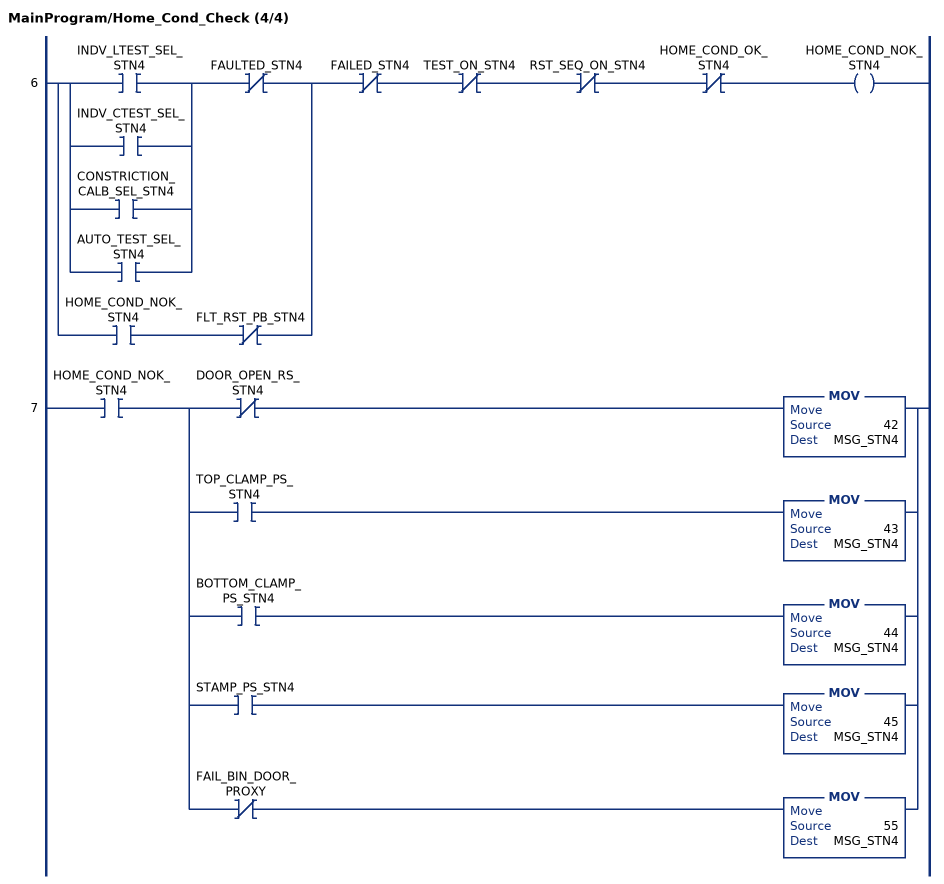
   6: [[XIC(INDV_LTEST_SEL_STN4) ,XIC(INDV_CTEST_SEL_STN4) ,XIC(CONSTRICTION_CALB_SEL_STN4) ,XIC(AUTO_TEST_SEL_STN4) ] XIO(FAULTED_STN4) ,XIC(HOME_COND_NOK_STN4) XIO(FLT_RST_PB_STN4) ]XIO(FAILED_STN4)XIO(TEST_ON_STN4)XIO(RST_SEQ_ON_STN4)XIO(HOME_COND_OK_STN4)OTE(HOME_COND_NOK_STN4);
   7: XIC(HOME_COND_NOK_STN4)[XIO(DOOR_OPEN_RS_STN4) MOV(42,MSG_STN4) ,XIC(TOP_CLAMP_PS_STN4) MOV(43,MSG_STN4) ,XIC(BOTTOM_CLAMP_PS_STN4) MOV(44,MSG_STN4) ,XIC(STAMP_PS_STN4) MOV(45,MSG_STN4) ,XIO(FAIL_BIN_DOOR_PROXY) MOV(55,MSG_STN4) ];
END_ROUTINE
